TYPE ST_Foo :
STRUCT
	bVal01	:	BOOL;
	bVal02	:	BOOL;
END_STRUCT
END_TYPE

(* stored: Version 1.1.0.1, ProductVersion 3.1.4020.6
   DUT ST_Foo: Id {486bfbcb-0ad2-4742-a33e-b99ad53a1691} *)
